// TwinCAT 3 PLC project Untitled1
// ProgramVersion: 3.1.4023.0
// libraries:
//   CmpBitmapPool, * (System)
//   Tc2_MC2, * (Beckhoff Automation GmbH)
//   Tc2_Standard, * (Beckhoff Automation GmbH)
//   Tc2_System, * (Beckhoff Automation GmbH)
//   Tc2_Utilities, * (Beckhoff Automation GmbH)
//   Tc3_Module, * (Beckhoff Automation GmbH)
// project tree:
//   DUTs/ A21ToolStorage.TcDUT (not stored), Bundle.TcDUT (not stored), EOAT.TcDUT (not stored), Interval.TcDUT (not stored), PositionMaterials.TcDUT (not stored)
//   DUTs/Enums/ A21.TcDUT (not stored), Chipboard.TcDUT (not stored), Homing.TcDUT (not stored), SectionEnum.TcDUT (not stored), Surface.TcDUT (not stored), WoodBunk.TcDUT
//   DUTs/Insertion/Drives/ AirPiston.TcPOU, ClearLinkMC.TcPOU (not stored), SimplePiston.TcPOU
//   DUTs/Insertion/ Insertion.TcPOU (not stored), SuctionPad.TcDUT (not stored)
//   DUTs/Insertion/Prototypes/ FBA_Drive.TcPOU (not stored), I_ContinuousDrive.TcIO (not stored), I_Drive.TcIO, I_PositionalDrive.TcIO, I_EncodedDrive.TcIO
//   DUTs/Machines/ Conveyor.TcPOU (not stored), ConveyorMode.TcDUT (not stored), KukaRobot.TcPOU, RobotA21.TcPOU, StrapMachine.TcPOU (not stored)
//   DUTs/Material Holders/ MaterialHolder.TcPOU, SkidMagazine.TcPOU (not stored), StagingTable.TcPOU, MaterialSlot.TcDUT (not stored)
//   GVLs/ StorageArrays.TcGVL, GVL.TcGVL, Hardware.TcGVL (not stored), Misc.TcGVL (not stored)
//   / PlcTask.TcTTO (not stored)
//   POUs/ FB_System.TcPOU (not stored), MAIN.TcPOU (not stored), WoodBunkEx.TcPOU, ChipboardEx.TcPOU (not stored)
//   POUs/Hardware Calls/ InsertionQuality.TcPOU (not stored), CallHardware.TcPOU (not stored), SetSuctions.TcPOU (not stored), SetupHardware.TcPOU
//   POUs/Utility/ AddToStringArray.TcPOU (not stored), BoolVLArrayToInteger.TcPOU (not stored), BoolPtrArrayToInteger.TcPOU (not stored), IntegerBitAccess.TcPOU (not stored), IntegerToBoolArray.TcPOU (not stored), JoinStrings.TcPOU (not stored), WithinTolerance.TcPOU (not stored)
// real-time tasks:
//   TASK PlcTask: cycle T#10ms, priority 20, ADS port 350

// ---- DUTs/Enums/WoodBunk.TcDUT
{attribute 'qualified_only'}
{attribute 'to_string'}
TYPE WoodBunk : //21
(
	NULL, 
	
	WDS08, //side
	WDS10, 
	WDS12, 
	WDS14, 
	
	WDS20, //side - same size as TOP
	WDS22, 
	WDS28, 
	
	WDB20, //bottom
	WDB22, 
	WDB28,

	WDT20, //top
	WDT22, 
	WDT28,
	
	WDW20, //special top (wide) 
	WDW22,
	
	
	size
	(*
	WDS08_WDS08, //side combined - X - 2 wood bunks joined by underscore
	WDS08_WDS10, 
	WDS12_WDS12, 
	WDS12_WDS14, 
	WDS20_WDS10, 
	WDS20_WDS12, 
	
	sizeAll
	*)
);
END_TYPE

// ---- GVLs/StorageArrays.TcGVL
//{attribute 'qualified_only'}
VAR_GLOBAL //data arrays to be passed into material holder FBs - do not access directly
	
	skidSlotsA21Left, skidSlotsA21Right : ARRAY[1..2] OF STRING; //chipboard skid
	skidOccupancyA21Left, skidOccupancyA21Right : ARRAY[1..2] OF BOOL;
	skidHmiA21Left, skidHmiA21Right : ARRAY[1..2] OF MaterialSlot;
	
	magazineSlotsA21Left, magazineSlotsA21Right : ARRAY[1..15] OF STRING; //wood bunk magazine
	magazineOccupancyA21Left, magazineOccupancyA21Right : ARRAY[1..15] OF BOOL;
	magazineHmiA21Left, magazineHmiA21Right : ARRAY[1..15] OF MaterialSlot;
	
	tableSlotsA21Left, tableSlotsA21Right : ARRAY[1..10] OF STRING; //staging table
	tableOccupancyA21Left, tableOccupancyA21Right AT %I* : ARRAY[1..10] OF BOOL;
	tableHmiA21Left, tableHmiA21Right : ARRAY[1..10] OF MaterialSlot;
END_VAR

// ---- GVLs/GVL.TcGVL
{attribute 'qualified_only'}
VAR_GLOBAL CONSTANT
	maxPairs : INT := 16;
	maxQueue : INT := 16;
END_VAR

// ---- DUTs/Insertion/Prototypes/I_Drive.TcIO
INTERFACE I_Drive

{attribute 'monitoring':='call'}
PROPERTY ABSTRACT AtHome : BOOL
GET
END_GET
END_PROPERTY

{attribute 'monitoring':='call'}
PROPERTY ABSTRACT AtInnerLimit : BOOL
GET
END_GET
END_PROPERTY

{attribute 'monitoring':='call'}
PROPERTY ABSTRACT AtOuterLimit : BOOL
GET
END_GET
END_PROPERTY

{attribute 'monitoring':='call'}
PROPERTY ABSTRACT Busy : BOOL
GET
END_GET
END_PROPERTY

{attribute 'monitoring':='call'}
PROPERTY ABSTRACT Contact : BOOL
GET
END_GET
END_PROPERTY

{attribute 'monitoring':='call'}
PROPERTY ABSTRACT Error : BOOL
GET
END_GET
END_PROPERTY

{attribute 'monitoring':='call'}
PROPERTY ABSTRACT HomeSet : BOOL
GET
END_GET
END_PROPERTY

METHOD ABSTRACT homingSequence : BOOL
VAR_INPUT
END_VAR
END_METHOD

METHOD ABSTRACT stop : BOOL
VAR_INPUT
END_VAR
END_METHOD

END_INTERFACE

// ---- DUTs/Insertion/Prototypes/I_PositionalDrive.TcIO
INTERFACE I_PositionalDrive EXTENDS I_Drive

PROPERTY ABSTRACT CurrentPosition : LREAL
GET
END_GET
SET
END_SET
END_PROPERTY

METHOD ABSTRACT moveAbsolute : BOOL
VAR_INPUT
	newTarget : LREAL; 
END_VAR
END_METHOD

METHOD ABSTRACT moveRelative : BOOL
VAR_INPUT
	distance : LREAL;
END_VAR
END_METHOD

PROPERTY ABSTRACT TargetPosition : LREAL
GET
END_GET
SET
END_SET
END_PROPERTY

END_INTERFACE

// ---- DUTs/Insertion/Prototypes/I_EncodedDrive.TcIO
INTERFACE I_EncodedDrive EXTENDS I_PositionalDrive, I_ContinuousDrive
//this drive can perform absolute/relative targeting and continuous motion
//only used if a drive with both encoded and continuous behavior is needed

END_INTERFACE

// ---- DUTs/Insertion/Drives/AirPiston.TcPOU
FUNCTION_BLOCK AirPiston EXTENDS FBA_Drive IMPLEMENTS I_ContinuousDrive
VAR_OUTPUT
	valveExtend AT %Q* : BOOL;
	valveRetract AT %Q* : BOOL;
END_VAR
VAR
	mode : (HOLD, IN, OUT, BRAKE);
	
	useBrake : BOOL; //set to FALSE if retraction brake is not required
	brakePulse : TP; //generates the retraction pulse
END_VAR
VAR_STAT CONSTANT
	brakeTime : TIME := T#650MS;
END_VAR

IF NOT bEnable THEN
	stop();
	RETURN;
END_IF

brakePulse(IN:= , PT:= brakeTime, Q=> , ET=> ); //reversal to act as brake
brakePulse.IN := brakePulse.IN AND brakePulse.Q; //automatically turn off pulse

override(); //alters the mode to prevent exceeding limits

CASE mode OF
	HOLD:
		valveExtend := FALSE;
		valveRetract := FALSE;
		
	IN:
		valveExtend := TRUE;
		valveRetract := FALSE;
		
	OUT:
		valveExtend := FALSE;
		valveRetract := TRUE;
		
	BRAKE: //coasts past inner limit, then slides back
		valveExtend := FALSE;
		valveRetract := TRUE;
		
		IF innerLimit THEN
			mode := HOLD;
		END_IF
		
END_CASE

valveRetract := valveRetract OR brakePulse.Q; //from mode or brake

PROPERTY Busy : BOOL
GET
Busy :=
	mode <> HOLD AND
	valveExtend OR valveRetract;
END_GET
END_PROPERTY

PROPERTY Error : BOOL
GET
END_GET
END_PROPERTY

METHOD extend : BOOL
VAR_INPUT
END_VAR
IF mode <> BRAKE THEN
	mode := IN;
END_IF
END_METHOD

METHOD homingSequence : BOOL
CASE step OF
	Homing.IDLE:
		step := Homing.OUT;
		
	Homing.OUT: //towards home
		mode := OUT;
		
		IF home THEN //if reached home
			step := Homing.DONE;
		END_IF
		
	Homing.DONE:
		mode := HOLD;
		homingComplete := TRUE;
		
		homingSequence := TRUE;		
	
END_CASE
END_METHOD

METHOD moveContinuous : BOOL
VAR_INPUT
	direction : MC_Direction;
END_VAR
IF direction = MC_Positive_Direction THEN
	retract();
ELSIF direction = MC_Negative_Direction THEN
	extend();
END_IF
END_METHOD

METHOD PRIVATE override : BOOL
VAR_INPUT
END_VAR
IF brakePulse.Q THEN
	mode := HOLD;
END_IF

IF home AND_THEN (valveRetract OR mode = OUT) THEN
	mode := HOLD;
	
ELSIF (innerLimit OR contactSensor) AND_THEN (valveExtend OR mode = IN) THEN	
	brakePulse.IN := useBrake;
	mode := HOLD;
END_IF


IF NOT bEnable THEN
	stop();
END_IF
END_METHOD

METHOD retract : BOOL
VAR_INPUT
END_VAR
IF mode <> BRAKE THEN
	mode := OUT;
END_IF
END_METHOD

METHOD stop : BOOL
VAR_INPUT
END_VAR
valveExtend := FALSE;
valveRetract := FALSE;
mode := HOLD;
END_METHOD

END_FUNCTION_BLOCK

// ---- DUTs/Insertion/Drives/SimplePiston.TcPOU
FUNCTION_BLOCK SimplePiston
VAR_INPUT
	bEnable : BOOL;
END_VAR
VAR_OUTPUT
	pistonExtend AT %Q* : BOOL;
	pistonRetract AT %Q* : BOOL;
	
	extended AT %I* : BOOL;
	retracted AT %I* : BOOL;
END_VAR
VAR
	mode : (HOLD, IN, OUT);
END_VAR

IF
	NOT bEnable OR
	(retracted AND_THEN (pistonRetract OR mode = OUT)) OR
	(extended AND_THEN (pistonExtend OR mode = IN))
THEN
	mode := HOLD;
END_IF

CASE mode OF
	HOLD:
		pistonRetract := FALSE;
		pistonExtend := FALSE;
		
	IN:
		pistonRetract := FALSE;
		pistonExtend := TRUE;
	
	OUT:
		pistonRetract := TRUE;
		pistonExtend := FALSE;
	
END_CASE

METHOD extend : BOOL
VAR_INPUT
END_VAR
mode := IN;
END_METHOD

METHOD retract : BOOL
VAR_INPUT
END_VAR
mode := OUT;

retract := retracted;
END_METHOD

METHOD stop : BOOL
VAR_INPUT
END_VAR
pistonExtend := FALSE;
pistonRetract := FALSE;
mode := HOLD;
END_METHOD

END_FUNCTION_BLOCK

// ---- DUTs/Machines/KukaRobot.TcPOU
FUNCTION_BLOCK KukaRobot
VAR_OUTPUT
	forceStop AT %Q* : BOOL;
	resetSignal AT %Q* : BOOL;
	
	offline AT %I* : BOOL;
	operational : BOOL;
	reservation : INT := SectionEnum.NULL_SECTION;
	
	error : BOOL;
	errId : DINT;
	
	outputs AT %Q* : ARRAY[1..50] OF WORD;
	inputs AT %I* : ARRAY[1..20] OF WORD;
END_VAR
VAR
	hmiReservation : STRING;
END_VAR
(*
generic KUKA robot with 50 WORD outputs and 20 WORD inputs
includes minimal diagnostics to detect if robot is offline
robots should always be reserved before sending a task
*)

operational := NOT offline;

error := offline; //add any addition conditions with OR

//{attribute 'monitoring' := 'variable'}
{attribute 'monitoring' := 'call'}
PROPERTY Busy : BOOL
GET
END_GET
END_PROPERTY

METHOD clearCommand : BOOL
VAR_INPUT
END_VAR
MEMSET(ADR(outputs), 0, SIZEOF(outputs));
END_METHOD

//{attribute 'monitoring' := 'variable'}
{attribute 'monitoring' := 'call'}
PROPERTY Done : BOOL
GET
END_GET
END_PROPERTY

METHOD eStop : BOOL
VAR_INPUT
END_VAR
forceStop := TRUE;
eStop := TRUE;
END_METHOD

METHOD fullCommand : BOOL
VAR_INPUT
	newOutputs : REFERENCE TO ARRAY[1..50] OF WORD;
END_VAR
//IF NOT Busy THEN
	//RETURN;
//END_IF

outputs := newOutputs;
fullCommand := Done;

(*
CASE step OF
	SEND_COMMAND: //wait 1 cycle
		outputs := newOutputs;
		step := WAIT;
		
	WAIT:
		IF done THEN
			(*	
			IF NOT reset() THEN
				RETURN;
			END_IF
			
			step := 0;
			*)
			setCommandAndWait := TRUE;
		END_IF
		
END_CASE
*)
END_METHOD

{attribute 'monitoring' := 'call'}
PROPERTY Ready : BOOL
GET
END_GET
END_PROPERTY

METHOD release : BOOL
VAR_INPUT
	reservee : INT;
END_VAR
IF reservation = reservee THEN
	reservation := SectionEnum.NULL_SECTION;
	release := TRUE;
END_IF
END_METHOD

METHOD reserve : BOOL
VAR_INPUT
	reservee : INT;
END_VAR
(*
this method exists because chipboard and wood bunk operations use the same robot
both sections need to check if the robot is open to commands before use
*)
IF Reserved AND reservation = reservee THEN
	reserve := TRUE;

ELSIF NOT Reserved THEN
	reservation := reservee;
	reserve := TRUE;

END_IF
END_METHOD

{attribute 'monitoring' := 'call'}
PROPERTY Reserved : BOOL
GET
Reserved := reservation <> SectionEnum.NULL_SECTION;
END_GET
END_PROPERTY

METHOD reset : BOOL
//resetSignal := TRUE;
//done := FALSE;

MEMSET(ADR(outputs), 0, SIZEOF(outputs));
(*
IF ready AND completedTask = 0 THEN
	resetSignal := FALSE;
	reset := TRUE;
END_IF
*)
END_METHOD

METHOD resume : BOOL
VAR_INPUT
END_VAR
forceStop := FALSE;

resume := NOT error AND errId = 0;
END_METHOD

METHOD setGroup : BOOL
VAR_INPUT
	group : INT;
	value : INT;
END_VAR
{warning disable C0195}
outputs[group] := value;
END_METHOD

END_FUNCTION_BLOCK

// ---- DUTs/Machines/RobotA21.TcPOU
FUNCTION_BLOCK RobotA21 EXTENDS KukaRobot
VAR_OUTPUT //from outputs array
	{warning disable C0195}
	taskID : A21;
	param1 : INT;
	param2 : INT;
	Xmm : INT;
	Ymm : INT;
	Zmm : INT;
	angle : INT;
	stagingOccupancy : INT;
	insertionSuctionStatus : INT;
	magazineStatus : INT; //unused
	inspectionValue : INT;
	
	strapSafetyOut : BOOL;
END_VAR
VAR_OUTPUT //from inputs array
	tool : SectionEnum := SectionEnum.WOOD_BUNK;
	suspendedMaterial : STRING;
	//gripper : EOAT := (id := SectionEnum.WOOD_BUNK, material := '');
	
	completedTask : A21;
	eoatDistance : INT;
	woodBunkAvailability : INT;
	chipboardAvailability : INT;
	materialAtHoldingPosition : INT;
	
	strapSafetyIn : BOOL;
END_VAR
VAR
	reservationEnum : SectionEnum;
	hmiTask : STRING;
	hmiTool : STRING;
END_VAR
(*
extends KukaRobot
assigns descriptive labels to each IO group from the array
additional section-specific methods to get/set IO groups
*)

(*
parameters - aliases to IO elements
command - full IO array
*)
{warning disable C0195}
SUPER^();

strapSafetyOut := NOT strapperA21.enable AND NOT strapperA21.execute;
outputs[8].15 := strapSafetyOut;

outputs[1] := taskID;
outputs[2] := param1;
outputs[3] := param2;
outputs[4] := Xmm;
outputs[5] := Ymm;
outputs[6] := Zmm;
outputs[7] := angle;
outputs[8] := stagingOccupancy;
outputs[9] := insertionSuctionStatus;
outputs[10] := magazineStatus;
outputs[11] := inspectionValue;

outputs[8].15 := strapSafetyOut;

refreshParameters();

reservationEnum := reservation;
IF reservationEnum = SectionEnum.NULL_SECTION THEN
	hmiReservation := 'N/A';
ELSE
	hmiReservation := TO_STRING(reservationEnum);
END_IF

hmiTask := TO_STRING(taskID);
hmiTool := TO_STRING(tool);

{attribute 'monitoring' := 'call'}
PROPERTY Busy : BOOL
GET
VAR
	//emptyOutput : ARRAY[1..50] OF INT;
END_VAR
//Busy stays TRUE until outputs are cleared AND completed task has elapsed
//Ready is always inverse of Busy
refreshParameters();

Busy := taskID <> 0 OR completedTask <> 0;
END_GET
END_PROPERTY

METHOD changeEOAT : BOOL
VAR_INPUT
	targetTool : SectionEnum;
END_VAR
setGroup(group := 1, value := A21.TOOL_CHANGE_CHIPBOARD);
setGroup(group := 1, value := A21.TOOL_CHANGE_BUNK);

changeEOAT := tool = targetTool;
END_METHOD

METHOD clearCommand : BOOL
VAR_INPUT
END_VAR
SUPER^.clearCommand();

refreshParameters();
END_METHOD

{attribute 'monitoring' := 'call'}
PROPERTY Done : BOOL
GET
refreshParameters();

Done :=
	completedTask = taskID AND
	taskID <> 0 AND
	completedTask <> 0;
END_GET
END_PROPERTY

{attribute 'monitoring' := 'call'}
PROPERTY HoldMaterial : STRING
GET
HoldMaterial := suspendedMaterial;
END_GET
SET
suspendedMaterial := HoldMaterial;
END_SET
END_PROPERTY

{attribute 'monitoring' := 'call'}
PROPERTY Ready : BOOL
GET
refreshParameters();

Ready := taskID = 0 AND completedTask = 0;
END_GET
END_PROPERTY

METHOD PRIVATE refreshParameters : BOOL
VAR_INPUT
END_VAR
{warning disable C0196}
taskID := outputs[1];
param1 := outputs[2];
param2 := outputs[3];
Xmm := outputs[4];
Ymm := outputs[5];
Zmm := outputs[6];
angle := outputs[7];
stagingOccupancy := outputs[8];
insertionSuctionStatus := outputs[9];
magazineStatus := outputs[10]; //unused
inspectionValue := outputs[11];

completedTask := inputs[1];
eoatDistance := inputs[2];
woodBunkAvailability := inputs[3];
chipboardAvailability := inputs[4];
materialAtHoldingPosition := inputs[5];
//robotEOAT := inputs[6];

strapSafetyIn := inputs[4].15;
END_METHOD

METHOD setGroup : BOOL
VAR_INPUT
	group : INT;
	value : INT;
END_VAR
SUPER^.setGroup(group := group, value := value);

refreshParameters();
END_METHOD

METHOD setParameters : BOOL
VAR_INPUT
	newTaskID : INT;
	newParam1 : INT;
	newParam2 : INT;
	newXmm : INT;
	newYmm : INT;
	newZmm : INT;
	newAngle : INT;
	newStagingOccupancy : INT;
	newInsertionSuctionStatus : INT;
	newMagazineStatus : INT; //unused
	newInspectionValue : INT;
END_VAR
setGroup(group := 1, value := newTaskID);
setGroup(group := 2, value := newParam1);
setGroup(group := 3, value := newParam2);
setGroup(group := 4, value := newXmm);
setGroup(group := 5, value := newYmm);
setGroup(group := 6, value := newZmm);
setGroup(group := 7, value := newAngle);

newStagingOccupancy.15 := NOT strapperA21.enable AND NOT strapperA21.execute;
setGroup(group := 8, value := newStagingOccupancy);

setGroup(group := 9, value := newInsertionSuctionStatus);
setGroup(group := 10, value := newMagazineStatus);
setGroup(group := 11, value := newInspectionValue);

refreshParameters();
END_METHOD

END_FUNCTION_BLOCK

// ---- DUTs/Material Holders/MaterialHolder.TcPOU
FUNCTION_BLOCK MaterialHolder
VAR_IN_OUT
	slots : ARRAY[*] OF STRING;
	occupied : ARRAY[*] OF BOOL;
	
	hmiTable : ARRAY[*] OF MaterialSlot;
END_VAR
VAR
	numSlots : INT;
END_VAR

(*
by default:
	hmiTable contains the true data, including IO mapped to hardware
	slots and occupied cyclically copy data from hmiTable

if hmiTable is NULL (not passed in), then slots and occupied will store the true data
	
the program will access data using slots/occupied via methods
when the data is changed, data is copied from slots/occupied to hmiTable

this ensures that the methods update the HMI, and the HMI updates the data
*)


IF hmiTable <> 0 AND_THEN (slots <> 0  AND occupied <> 0) THEN
	writeArrays();
END_IF

numSlots := TO_INT(UPPER_BOUND(slots, 1) - LOWER_BOUND(slots, 1) + 1);

METHOD clear : BOOL
VAR_INPUT
END_VAR
MEMSET(ADR(slots), 0, SIZEOF(slots));
END_METHOD

METHOD findSlot : BOOL
VAR_INPUT
	materialID : STRING;
END_VAR
VAR_OUTPUT
	atPosition : INT := -1;
END_VAR
VAR
	i : INT;
END_VAR
(*
IF materialID = '' THEN
	RETURN;
END_IF
*)
FOR i:=1 TO GVL.maxQueue BY 1 DO
	IF slots[i] = materialID THEN
		atPosition := i;
		findSlot := TRUE;
		RETURN;
	END_IF
END_FOR
END_METHOD

METHOD getSlot : STRING
VAR_INPUT
	i : DINT;
END_VAR
VAR_OUTPUT
	errorBounds : BOOL;
END_VAR
errorBounds := i < LOWER_BOUND(slots, 1) OR i > UPPER_BOUND(slots, 1);

IF errorBounds THEN
	RETURN;
END_IF

getSlot := slots[i];
END_METHOD

METHOD getSlotsAsArray : POINTER TO STRING
getSlotsAsArray := ADR(slots);
END_METHOD

METHOD isOccupied : BOOL
VAR_INPUT
	i : DINT;
END_VAR
VAR_OUTPUT
	errorBounds : BOOL;
END_VAR
errorBounds := i < LOWER_BOUND(slots, 1) OR i > UPPER_BOUND(slots, 1);

IF errorBounds THEN
	RETURN;
END_IF

isOccupied := occupied[i];
END_METHOD

METHOD setSlots : BOOL
VAR_IN_OUT
	newSlots : ARRAY[*] OF STRING;
END_VAR
VAR
	i : DINT;
	j : DINT;
END_VAR
{warning disable C0195}
setSlots := MEMCPY(
	slots, 
	newSlots, 
	SIZEOF(STRING) * MIN(
		(1 + UPPER_BOUND(newSlots, 1) - LOWER_BOUND(newSlots, 1)),
		(1 + UPPER_BOUND(slots, 1) - LOWER_BOUND(slots, 1))
	)) > 0;
	
IF hmiTable <> 0 THEN
	writeHmiTable();
END_IF
END_METHOD

METHOD PROTECTED writeArrays : BOOL
VAR
	i : DINT;
END_VAR
FOR i:=LOWER_BOUND(hmiTable, 1) TO UPPER_BOUND(hmiTable, 1) BY 1 DO
	slots[i] := hmiTable[i].material;
	occupied[i] := hmiTable[i].occupied;
END_FOR
END_METHOD

METHOD PROTECTED writeHmiTable : BOOL
VAR
	i : DINT;
END_VAR
FOR i:=LOWER_BOUND(hmiTable, 1) TO UPPER_BOUND(hmiTable, 1) BY 1 DO
	hmiTable[i].material := slots[i];
	hmiTable[i].occupied := occupied[i];
END_FOR
END_METHOD

END_FUNCTION_BLOCK

// ---- DUTs/Material Holders/StagingTable.TcPOU
FUNCTION_BLOCK StagingTable EXTENDS MaterialHolder

SUPER^();

METHOD autofill : BOOL
VAR_INPUT
	materialID : STRING;
END_VAR
VAR_OUTPUT
	slot : INT;
END_VAR
VAR
	i : INT;
END_VAR
(*
this method will automatically find an open slot
*)
IF isFull() OR materialID = '' THEN
	RETURN;
END_IF

IF findOpenSlot(materialID, openSlot=> slot) THEN
	place(slot, materialID);
	autofill := TRUE;
END_IF

IF hmiTable <> 0 THEN
	writeHmiTable();
END_IF
END_METHOD

METHOD findOpenSlot : BOOL
VAR_INPUT
	materialID : STRING;
END_VAR
VAR_OUTPUT
	openSlot : INT := 0;
END_VAR
VAR
	i : INT;
END_VAR
IF FIND(materialID, 'WDW') > 0 THEN //top wide, load in slot 9-10
	FOR i:=9 TO 10 BY 1 DO
		IF slots[i] = '' THEN
			findOpenSlot := TRUE;
			openSlot := i;
			RETURN;
		END_IF
	END_FOR
	
//ELSIF FIND(materialID, 'WDT') > 0 OR FIND(materialID, 'WDS') > 0 THEN //standard width, load in slot 3-10
ELSIF FIND(materialID, 'WD') > 0 THEN //standard width, load in slot 1-8
	FOR i:=1 TO 8 BY 1 DO
		IF slots[i] = '' THEN
			findOpenSlot := TRUE;
			openSlot := i;
			RETURN;
		END_IF
	END_FOR
	
END_IF
END_METHOD

METHOD isEmpty : BOOL
VAR
	i : INT;
	temp : BOOL;
END_VAR
FOR i:=1 TO numSlots BY 1 DO
	temp := temp OR occupied[i]; //TRUE if any slots are occupied
END_FOR

isEmpty := NOT temp; //invert result - FALSE if any slots are occupied
END_METHOD

METHOD isFull : BOOL
VAR
	i : INT;
	temp : BOOL := TRUE;
END_VAR
FOR i:=1 TO numSlots BY 1 DO
	temp := temp AND occupied[i];
END_FOR

isFull := temp;
END_METHOD

METHOD place : BOOL
VAR_INPUT
	i : INT;
	materialID : STRING;
END_VAR
IF slots[i] = '' THEN
	slots[i] := materialID;
	place := TRUE;
END_IF

IF hmiTable <> 0 THEN
	writeHmiTable();
END_IF
END_METHOD

METHOD remove : BOOL
VAR_INPUT
	i : INT;
END_VAR
VAR_OUTPUT
	materialID : STRING;
END_VAR
remove := slots[i] <> '';

materialID := slots[i];
slots[i] := '';

IF hmiTable <> 0 THEN
	writeHmiTable();
END_IF
END_METHOD

END_FUNCTION_BLOCK

// ---- POUs/Hardware Calls/SetupHardware.TcPOU
FUNCTION SetupHardware : BOOL
VAR
	iWoodBunkSlot : WoodBunk;
	iChipboardSlot : Chipboard;
	
	slotsArr : ARRAY[1..GVL.maxQueue] OF STRING;
	
	i : INT;
END_VAR

FOR iWoodBunkSlot:=1 TO WoodBunk.size-1 BY 1 DO //init wood bunk magazine slots
	magazineA21Left.setSlot(i := iWoodBunkSlot, material := TO_STRING(iWoodBunkSlot), error => );
	magazineA21Right.setSlot(i := iWoodBunkSlot, material := TO_STRING(iWoodBunkSlot), error => );
END_FOR

//--------------------------------------------------

FOR iChipboardSlot:=1 TO Chipboard.size-1 BY 1 DO //init chipboard skid slots
	skidA21Left.setSlot(i := iChipboardSlot, material := TO_STRING(iChipboardSlot), error => );
	skidA21Right.setSlot(i := iChipboardSlot, material := TO_STRING(iChipboardSlot), error => );
END_FOR

//--------------------------------------------------

FOR i:=1 TO GVL.maxQueue BY 1 DO //get wood bunk magazine + chipboard skid availability from robot1 and robot2
	{warning disable C0195}
	skidA21Left.setOccupancy( i := i, occupancy := IntegerBitAccess(robot1.inputs[4], i-1) );
	skidA21Right.setOccupancy( i := i, occupancy := IntegerBitAccess(robot2.inputs[4], i-1) );

	magazineA21Left.setOccupancy( i := i, occupancy := IntegerBitAccess(robot1.inputs[3], i-1) );
	magazineA21Right.setOccupancy( i := i, occupancy := IntegerBitAccess(robot2.inputs[3], i-1) );
END_FOR

//--------------------------------------------------

//enable all drives
verticalDriveA21Left.bEnable := 
verticalDriveA21Right.bEnable := 
horizontalDriveA21Left.bEnable := 
horizontalDriveA21Right.bEnable := 
pistonA21Bottom.bEnable := 
TRUE;

END_FUNCTION

// ---- POUs/WoodBunkEx.TcPOU
FUNCTION_BLOCK WoodBunkEx
VAR_IN_OUT //controls
	execute : BOOL;
	stop : BOOL;
	
	manualStep : BOOL;
	manualSuction : BOOL;
END_VAR
VAR_IN_OUT //references to required hardware
	robotLeft, robotRight : RobotA21;
	toolStorageLeft, toolStorageRight : A21ToolStorage;
	
	stagingTableLeft, stagingTableRight : StagingTable;
	magazineLeft, magazineRight : SkidMagazine;
	
	strapper : StrapMachine;
	
	horizontalDriveLeft, horizontalDriveRight : AirPiston;
	verticalDriveLeft, verticalDriveRight : ClearLinkMC;
	pistonBottom : SimplePiston;
	
	suctionTop : ARRAY[*] OF SuctionPad; (*1..3*)
	suctionLeft : ARRAY[*] OF SuctionPad; (*1..4*)
	suctionRight : ARRAY[*] OF SuctionPad; (*1..4*)
	suctionBottom : ARRAY[*] OF SuctionPad; (*1..2*)
END_VAR
VAR_OUTPUT
	//ready : BOOL;
	done : BOOL;
	
	generalError : BOOL;
	errorLeft, errorRight : BOOL;
END_VAR
VAR //for testing, to be removed when deployoed
	latchLeft, latchRight : BOOL; //prevents SMC sliders from overshooting the inner limit sensor
	
	suctionEnableTop : BOOL;
	suctionEnableLeft : BOOL;
	suctionEnableRight : BOOL;
	suctionEnableBottom : BOOL;
END_VAR
VAR	
	topSuctionDelay : TON;
	
	step : (IDLE, STAGING, LOAD_WB, PUSH, STRAP, RELEASE, COMPLETE := 1050);
	iPair : INT;
	//these 2 ints should replace the 4 ints after
	masterStep : INT;
	subStepLeft, subStepRight : INT;
	
	loadSet : INT;
	loadStepLeft, loadStepRight : INT;
	
	stageSet : INT;	
	stageStepLeft, stageStepRight : INT;
	iSlotLeft, iSlotRight : INT;
END_VAR
VAR //local types
	demoHeight : REAL := 600; //mm
	materialsArr : ARRAY[0..GVL.maxPairs] OF PositionMaterials := [
		(
			position := 0,
			top := 'WDS20', left := 'WDS20', right := 'WDS20', bottom := 'WDB20'
		),
		(
			position := 69,
			top := 'WDS20', left := 'WDS20', right := 'WDS20', bottom := 'WDB20'
		)];
	
	templateSlotsLeft, templateSlotsRight : ARRAY[1..10] OF STRING;
	templateOccupancyLeft, templateOccupancyRight : ARRAY[1..10] OF BOOL;
	stagingTemplateLeft, stagingTemplateRight AT %M* : StagingTable;	
	stagingArrayLeft, stagingArrayRight : ARRAY[0..(GVL.maxPairs+1)*2] OF STRING;
	
	insertionLeft, insertionRight : Insertion;
	loadedMaterials : ARRAY[Surface.TOP..Surface.BOTTOM] OF STRING;
END_VAR
VAR CONSTANT
	sectionID : SectionEnum := SectionEnum.WOOD_BUNK;
END_VAR
VAR
	a,b,c,d : BOOL;
	suctionTimerLeft, suctionTimerRight : TON;
END_VAR

callLocalModules(); //initialize local modules

IF stop THEN
	stopSequence(); //stop everything
	RETURN;
END_IF

IF NOT insertionLeft.screw.HomeSet AND insertionRight.screw.HomeSet THEN
	homingSequence(); //homing all motion devices and robots
	RETURN;
END_IF

a S= suctionTop[1].occupied AND suctionTop[2].occupied AND suctionTop[3].occupied;
b S= suctionLeft[1].occupied AND suctionLeft[2].occupied AND suctionLeft[3].occupied AND suctionLeft[4].occupied;
c S= suctionRight[1].occupied AND suctionRight[2].occupied AND suctionRight[3].occupied AND suctionRight[4].occupied;
d S= suctionBottom[1].occupied AND suctionBottom[2].occupied;

CASE step OF
	IDLE:
		IF execute THEN
			execute := FALSE;
			suctionEnableTop := suctionEnableLeft := suctionEnableRight := suctionEnableBottom := FALSE;
			step := STAGING;
		END_IF
		
		SetSuctions(suctionTop, suctionEnableTop);
		SetSuctions(suctionLeft, suctionEnableLeft);
		SetSuctions(suctionRight, suctionEnableRight);
		SetSuctions(suctionBottom, suctionEnableBottom);
		
	STAGING:
		IF NOT done THEN
			done := stage(error => generalError);
		END_IF
		
		IF
			(manualStep AND_THEN execute) OR
			(NOT manualStep AND_THEN done)
		THEN
			execute := FALSE;
			done := FALSE;
			step := LOAD_WB;
		END_IF
	
	LOAD_WB:
		IF NOT done THEN
			done := load(pairIndex := iPair, error => generalError);
		END_IF
		
		IF manualSuction THEN
			SetSuctions(suctionTop, suctionEnableTop);
			SetSuctions(suctionLeft, suctionEnableLeft);
			SetSuctions(suctionRight, suctionEnableRight);
			SetSuctions(suctionBottom, suctionEnableBottom);
		END_IF
		
		IF
			(manualStep AND_THEN execute) OR
			(NOT manualStep AND_THEN done)
		THEN
			done := FALSE;
			suctionEnableTop := suctionEnableLeft := suctionEnableRight := suctionEnableBottom := FALSE;
			execute := FALSE;
			
			step := PUSH;
		END_IF
		
	PUSH:
		IF
			(manualStep AND_THEN execute) OR
			(latchLeft AND latchRight AND pistonBottom.extended)
		THEN
			latchLeft := latchRight := FALSE;
			execute := FALSE;
			step := STRAP;
		END_IF
		
		IF NOT validateSuctionQuality(checkTop:= TRUE, checkLeft:= TRUE, checkRight:= FALSE, checkBottom:= FALSE) THEN
			generalError := TRUE;
			RETURN;
		END_IF
		(*
		IF 
			insertionLeft.sliderPos <> demoHeight/2 //OR 
			//insertionRight.sliderPos <> demoHeight/2 //OR 
			//NOT insertionBottom.contact
		THEN
			insertionLeft.slideAbsolute(demoHeight/2);
			//insertionRight.slideAbsolute(demoHeight/2);
			RETURN;
		END_IF
		*)
		
		IF insertionLeft.screw.AtInnerLimit THEN
			latchLeft := TRUE;
		ELSIF NOT latchLeft THEN
			insertionLeft.press();
		END_IF
		
		IF insertionRight.screw.AtInnerLimit THEN
			latchRight := TRUE;
		ELSIF NOT latchRight THEN
			insertionRight.press();
		END_IF
		pistonBottom.extend();
		
	STRAP:
		topSuctionDelay(IN:= , PT:= T#1S, Q=> , ET=> );
		
		strapper.bEnable := TRUE;
		IF strapper.done THEN
			topSuctionDelay.IN := FALSE;
			step := RELEASE;
			RETURN;
		END_IF
		
		IF topSuctionDelay.Q THEN
			SetSuctions(suctionTop, FALSE);
			SetSuctions(suctionLeft, FALSE);
			SetSuctions(suctionRight, FALSE);
			SetSuctions(suctionBottom, FALSE);
		ELSIF strapper.atBundleLevel THEN
			topSuctionDelay.IN := TRUE;
		END_IF
		
		IF strapper.ready THEN
			strapper.strap();
		END_IF
		
		IF execute THEN
			topSuctionDelay.IN := FALSE;
			execute := FALSE;
			step := RELEASE;
		END_IF
		
	RELEASE: //release command		
		//insertionLeft.slideAbsolute(0);
		//insertionRight.slideAbsolute(0);
		
		insertionLeft.release();
		insertionRight.release();
		pistonBottom.retract();
		
		IF 
			(insertionLeft.screw.AtHome AND insertionRight.screw.AtHome AND pistonBottom.retracted) OR
			execute
		THEN
			execute := FALSE;
			step := COMPLETE;
		END_IF
	
	COMPLETE:
		//reset everything
		iPair := (iPair + 1) MOD GVL.maxPairs;
		step := IDLE;
		a := b := c := d := FALSE;
END_CASE

ACTION callLocalModules:
{warning disable C0371}
stagingTemplateLeft(slots := templateSlotsLeft, occupied := templateOccupancyLeft);
stagingTemplateRight(slots := templateSlotsRight, occupied := templateOccupancyRight);

insertionLeft(
	enable:= TRUE, 
	slider:= verticalDriveLeft, 
	screw:= horizontalDriveLeft, 
	contact=> , 
	softContact=> , 
	busy=> , 
	error=> , 
	home=> , 
	homingComplete=> , 
	sliderPos=> );
	
insertionRight(
	enable:= TRUE, 
	slider:= verticalDriveRight, 
	screw:= horizontalDriveRight,  
	contact=> , 
	softContact=> , 
	busy=> , 
	error=> , 
	home=> , 
	homingComplete=> , 
	sliderPos=> );
END_ACTION

METHOD createStagingArrayLeft : BOOL
VAR
	remainingMaterial : STRING;
	splitMaterial : STRING;
	
	i : INT;
END_VAR
FOR i:=0 TO GVL.maxPairs BY 1 DO
	remainingMaterial := materialsArr[i].top;
	WHILE FIND(remainingMaterial, '_') > 0 DO
		splitCombinedMaterials(remainingMaterial, splitMaterial);
		IF splitMaterial <> '' THEN
			AddToStringArray(arr := stagingArrayLeft, newString := splitMaterial, numElements => , nextIndex => );
		END_IF
	END_WHILE
	
	IF remainingMaterial <> '' THEN
		AddToStringArray(arr := stagingArrayLeft, newString := remainingMaterial, numElements => , nextIndex => );
	END_IF
	
	
	remainingMaterial := materialsArr[i].left;
	WHILE FIND(remainingMaterial, '_') > 0 DO
		splitCombinedMaterials(remainingMaterial, splitMaterial);
		IF splitMaterial <> '' THEN
			AddToStringArray(arr := stagingArrayLeft, newString := splitMaterial, numElements => , nextIndex => );
		END_IF
	END_WHILE
	
	IF remainingMaterial <> '' THEN
		AddToStringArray(arr := stagingArrayLeft, newString := remainingMaterial, numElements => , nextIndex => );
	END_IF
END_FOR
END_METHOD

METHOD createStagingArrayRight : BOOL
VAR
	remainingMaterial : STRING;
	splitMaterial : STRING;
	
	i : INT;
END_VAR
FOR i:=0 TO GVL.maxPairs*2 BY 1 DO
	remainingMaterial := materialsArr[i].bottom;
	WHILE FIND(remainingMaterial, '_') > 0 DO
		splitCombinedMaterials(remainingMaterial, splitMaterial);
		IF splitMaterial <> '' THEN
			AddToStringArray(arr := stagingArrayRight, newString := splitMaterial, numElements => , nextIndex => );
		END_IF
	END_WHILE
	
	IF remainingMaterial <> '' THEN
		AddToStringArray(arr := stagingArrayRight, newString := remainingMaterial, numElements => , nextIndex => );
	END_IF
	
	
	
	remainingMaterial := materialsArr[i].right;
	WHILE FIND(remainingMaterial, '_') > 0 DO
		splitCombinedMaterials(remainingMaterial, splitMaterial);
		IF splitMaterial <> '' THEN
			AddToStringArray(arr := stagingArrayRight, newString := splitMaterial, numElements => , nextIndex => );
		END_IF
	END_WHILE
	
	IF remainingMaterial <> '' THEN
		AddToStringArray(arr := stagingArrayRight, newString := remainingMaterial, numElements => , nextIndex => );
	END_IF
END_FOR
END_METHOD

METHOD PROTECTED generateStagingTemplate : BOOL
VAR
	remainingMaterial : STRING;
	splitMaterial : STRING;
	
	i : INT;
END_VAR
VAR_STAT
	temp : INT;
END_VAR
createStagingArrayLeft();
createStagingArrayRight();

//AddToStringArray(arr := stagingArrayLeft, newString := 'WDB20', numElements =>, nextIndex => );

(*
iterate through all pairs and autofill the template
replace succesfully autofilled materials with empty string

when staging needs to be performed a 2nd time, autofilling empty strings is always unsuccessful
*)
FOR i:=0 TO GVL.maxPairs*2 BY 1 DO
	IF stagingTemplateLeft.autofill(materialID := stagingArrayLeft[i]) THEN
		stagingArrayLeft[i] := '';
	END_IF
	
	IF stagingTemplateRight.autofill(materialID := stagingArrayRight[i]) THEN
		stagingArrayRight[i] := '';
	END_IF
END_FOR

(*
stagingTemplateLeft.autofill(demoPairWB.top);
stagingTemplateLeft.autofill(demoPairWB.left);

stagingTemplateRight.autofill(demoPairWB.right);
stagingTemplateRight.autofill(demoPairWB.bottom);
*)

generateStagingTemplate := TRUE;
END_METHOD

ACTION homingSequence:
insertionLeft.homingSequence();
insertionRight.homingSequence();
pistonBottom.retract();
END_ACTION

METHOD PROTECTED load : BOOL
VAR_INPUT
	pairIndex : INT;
END_VAR
VAR_OUTPUT
	error : BOOL;
END_VAR
VAR
	pair : REFERENCE TO PositionMaterials REF= materialsArr[pairIndex];
END_VAR
{warning disable C0371}

IF robotLeft.error OR robotRight.error THEN
	error := TRUE;
	RETURN;
	
ELSIF NOT robotLeft.reserve(sectionID) OR NOT robotRight.reserve(sectionID) THEN //loading requires both robots be reserved together
	RETURN;
	
ELSIF //robots have wrong tool
	(robotLeft.tool <> sectionID AND_THEN NOT robotLeft.changeEOAT(targetTool := sectionID)) OR
	(robotRight.tool <> sectionID AND_THEN NOT robotRight.changeEOAT(targetTool := sectionID))
THEN
	RETURN;
END_IF

CASE loadSet OF
	0: //top and bottom
		IF 
			loadingSequence(
				robot:= robotLeft, 
				table:= stagingTableLeft, 
				loadStep:= loadStepLeft, 
				slot:= iSlotLeft,
				suctions:= suctionTop,
				suctionTimer:= suctionTimerLeft,
				surfaceID:= Surface.TOP, 
				material:= pair.top, 
				fail=> errorLeft)
			
			AND
			loadingSequence(
				robot:= robotRight,
				table:= stagingTableRight, 
				loadStep:= loadStepRight, 
				slot:= iSlotRight,
				suctions:= suctionBottom,
				suctionTimer:= suctionTimerRight,
				surfaceID:= Surface.BOTTOM, 
				material:= pair.bottom, 
				fail=> errorRight)
			
		THEN
			suctionTimerLeft.IN := suctionTimerRight.IN := FALSE;
			loadStepLeft := loadStepRight := 0;
			loadSet := 10;
		END_IF
		
	10: //sides
		IF
			loadingSequence(
				robot:= robotLeft, 
				table:= stagingTableLeft, 
				loadStep:= loadStepLeft, 
				slot:= iSlotLeft,
				suctions:= suctionLeft,
				suctionTimer:= suctionTimerLeft,
				surfaceID:= Surface.LEFT, 
				material:= pair.left, 
				fail=> errorLeft)
			
			AND
			loadingSequence(
				robot:= robotRight, 
				table:= stagingTableRight, 
				loadStep:= loadStepRight, 
				slot:= iSlotRight,
				suctions:= suctionRight,
				suctionTimer:= suctionTimerRight,
				surfaceID:= Surface.RIGHT, 
				material:= pair.right, 
				fail=> errorRight)
		THEN
			suctionTimerLeft.IN := suctionTimerRight.IN := FALSE;
			loadStepLeft := loadStepRight := 0;
			loadSet := COMPLETE;
		END_IF
		
	COMPLETE:
		suctionTimerLeft.IN := suctionTimerRight.IN := FALSE;
		
		loadSet := 0;
		loadStepLeft := loadStepRight := 0;
		
		robotLeft.release(sectionID);
		robotRight.release(sectionID);
		
		load := TRUE;
END_CASE
END_METHOD

METHOD loadingSequence : BOOL
VAR_IN_OUT
	robot : RobotA21;
	table : StagingTable;
	suctions : ARRAY[*] OF SuctionPad;
	loadStep : INT;
	slot : INT;
	
	suctionTimer : TON;
END_VAR
VAR_INPUT
	surfaceID : Surface;
	material : STRING;
END_VAR
VAR_OUTPUT
	fail : BOOL;
END_VAR
VAR
	recoveryMagazine : REFERENCE TO SkidMagazine;
	recoveryStageStep : REFERENCE TO INT;
	suctionDelay : TIME := T#2S;
END_VAR
{warning disable C0371}
IF material = '' THEN
	robot.clearCommand();
	loadingSequence := TRUE;
	RETURN;
END_IF

CASE loadStep OF
	0: //wait for robot
		robot.clearCommand();
		IF robot.Ready THEN
			loadStep := 10;
			slot := 0;
		END_IF
		
	10: //grab from table
		IF slot < 1 AND_THEN NOT table.findSlot(materialID := material, atPosition => slot) THEN 
			fail := TRUE;
			RETURN;
		END_IF
		
		IF NOT table.isOccupied(i := slot) AND table.getSlot(i := slot) <> '' THEN //move from table to robot gripper
			robot.HoldMaterial := table.getSlot(i := slot);
			table.remove(i := slot, materialID => );
		END_IF
		
		IF robot.Done THEN
			loadStep := COMPLETE;
			RETURN;
		ELSIF robot.materialAtHoldingPosition >= 1 AND robot.materialAtHoldingPosition <= 8 THEN
			loadStep := 20;
			RETURN;
		END_IF
		
		CASE surfaceID OF
			Surface.TOP: 					robot.setGroup(group := 1, value := A21.LOAD_BUNK_TOP); 
			Surface.LEFT, Surface.RIGHT: 	robot.setGroup(group := 1, value := A21.LOAD_BUNK_SIDE);
			Surface.BOTTOM: 				robot.setGroup(group := 1, value := A21.LOAD_BUNK_BOTTOM);
		END_CASE
		robot.setGroup(group := 2, value := slot); 
			
	20: //place to insertion
		IF robot.materialAtHoldingPosition > 0 AND robot.HoldMaterial <> '' THEN //move from gripper to insertion
			IF loadedMaterials[surfaceID] = '' THEN //transfer to insertion as is
				loadedMaterials[surfaceID] := robot.HoldMaterial;
			ELSE //join with existing material using underscore _
				loadedMaterials[surfaceID] := JoinStrings(loadedMaterials[surfaceID], robot.HoldMaterial, '_');
			END_IF
			robot.HoldMaterial := '';
		END_IF
		
		CASE surfaceID OF
			Surface.TOP, Surface.BOTTOM:
				SetSuctions(suctions, TRUE (*robot.materialAtHoldingPosition = 1 OR robot.materialAtHoldingPosition = 4*));
				
			Surface.LEFT, Surface.RIGHT:
				SetSuctions(suctions, TRUE (*robot.materialAtHoldingPosition = 2 OR robot.materialAtHoldingPosition = 3*));
				(*
				FOR i:=LOWER_BOUND(suctions, 1) TO UPPER_BOUND(suctions, 1) BY 1 DO
					
					IF i < UPPER_BOUND(suctions, 1)/2 THEN
						suctions[i].enable := robot.materialAtHoldingPosition = 2; //enable upper half suctions
					ELSE
						suctions[i].enable := robot.materialAtHoldingPosition = 3; //enable lower half suctions
					END_IF

				END_FOR
				*)
		END_CASE
		
		suctionTimer(IN:= , PT:= suctionDelay, Q=> , ET=> );
		suctionTimer.IN := TRUE;
		IF NOT suctionTimer.Q THEN
			RETURN;
		END_IF
		
		IF robot.Done THEN
			suctionTimer.IN := FALSE;
			loadStep := COMPLETE;
			RETURN;
		END_IF
		
		robot.setGroup(group := 9, value := robot.materialAtHoldingPosition);
	
	COMPLETE:
		robot.clearCommand();
		
		//check insertion quality
		suctionTimer(IN:= , PT:= suctionDelay, Q=> , ET=> );
		suctionTimer.IN := TRUE;
		IF NOT suctionTimer.Q THEN
			RETURN;
		END_IF
		
		IF InsertionQuality(suctions := suctions, insertionMaterial := loadedMaterials[surfaceID], recipeMaterial := material) THEN
			loadingSequence := TRUE;
		ELSE //recovery - restage a new bunk to <slot> and reload
			suctionTimer.IN := FALSE;
			loadStep := 100;
			
		END_IF
		
	100: //recovery - restage and reload
		CASE surfaceID OF
			Surface.TOP, Surface.LEFT:
				recoveryMagazine REF= magazineLeft;			
				recoveryStageStep REF= stageStepLeft;
				
			Surface.RIGHT, Surface.BOTTOM:
				recoveryMagazine REF= magazineRight;			
				recoveryStageStep REF= stageStepRight;
				
		END_CASE
		
		IF
			stageSingle(
				robot:= robot, 
				table:= table, 
				magazine:= recoveryMagazine, 
				stageStep:= recoveryStageStep, 
				slot:= slot, 
				material:= material, 
				fail=> fail)
		THEN
			SetSuctions(suctionPads := suctions, state := FALSE);
			loadStep := 0; //retry
		END_IF
	
END_CASE
END_METHOD

METHOD splitCombinedMaterials : BOOL
VAR_IN_OUT
	materialID : STRING;
	splitMaterial : STRING;
END_VAR
VAR
	i : INT;
END_VAR
FindAndSplitChar(
	sSeparatorChar:= '_', 
	pSrcString:= ADR(materialID), 
	
	pLeftString:= ADR(splitMaterial), 
	nLeftSize:= SIZEOF(splitMaterial), 
	
	pRightString:= ADR(materialID), 
	nRightSize:= SIZEOF(materialID), 
	
	bSearchFromRight:= FALSE);
END_METHOD

METHOD stage : BOOL
VAR_OUTPUT
	error : BOOL;
END_VAR
{warning disable C0371}

CASE stageSet OF
	0: //create staging template
		IF generateStagingTemplate() THEN
			stageSet := 10;
		END_IF
	
	10: //staging sequence
		IF
			stagingSequence(				
				robot:= robotLeft, 
				template:= stagingTemplateLeft,
				table:= stagingTableLeft,  
				magazine:= magazineLeft, 
				stageStep:= stageStepLeft, 
				iSlot:= iSlotLeft,
				error=> errorLeft)
			
			AND
			stagingSequence(
				robot:= robotRight, 
				template:= stagingTemplateRight, 
				table:= stagingTableRight, 
				magazine:= magazineRight, 
				stageStep:= stageStepRight, 
				iSlot:= iSlotRight,
				error=> errorRight)
		THEN
			stageStepLeft := stageStepRight := 0;
			iSlotLeft := iSlotRight := 0;
			
			stageSet := COMPLETE;
		END_IF
		
	COMPLETE:
		stagingTemplateRight.clear(); //clear the staging templates
		stagingTemplateLeft.clear();
		
		robotLeft.release(sectionID); //release the robots
		robotRight.release(sectionID);
		
		stageSet := 0;
		stage := TRUE;
		
END_CASE
END_METHOD

METHOD stageSingle : BOOL
VAR_IN_OUT
	robot : RobotA21;
	table : StagingTable;
	magazine : SkidMagazine;
	stageStep : INT;
END_VAR
VAR_INPUT
	slot : INT;
	material : STRING;
END_VAR
VAR_OUTPUT
	fail : BOOL;
END_VAR
VAR
	column : INT; //valid positions start from 1
END_VAR
VAR CONSTANT
	suctionDistance : INT := 10;
END_VAR
{warning disable C0371}
{warning disable C0195}
(*
this method allows the staging of single bunks without the use of a template
neccessary for restaging bunks that are not loaded properly into insertions
*)

IF
	material = '' OR_ELSE
	table.getSlot(i := slot) = material
THEN
	robot.clearCommand();
	stageSingle := TRUE;
	RETURN;
END_IF

//follow the template as is
CASE stageStep OF
	0:
		robot.clearCommand();
		IF robot.Ready THEN
			stageStep := 10;
		END_IF
		
	10: //grab from magazine
		IF NOT magazine.findSlot(materialID := material, atPosition => column) THEN
			fail := TRUE;
			RETURN;
		END_IF
		
		IF robot.eoatDistance < suctionDistance THEN //robot is grabbing material
			robot.HoldMaterial := magazine.getSlot(i := column);
		END_IF
		
		IF robot.Done THEN
			stageStep := COMPLETE;
			RETURN;
		ELSIF table.isOccupied(slot) THEN //wood bunk registered on table
			stageStep := 20;
			RETURN;
		END_IF
		
		robot.setGroup(group := 1, value := A21.STAGE_BUNK);
		robot.setGroup(group := 2, value := column);
		robot.setGroup(group := 3, value := slot);
	
	20: //place to table
		IF
			table.isOccupied(slot) AND //staging table slot is occupied
			table.getSlot(slot) = '' AND //staging table has not recorded a bunk
			robot.HoldMaterial <> '' //robot is carrying a bunk
		THEN //move material from robot to table
			table.place(i := slot, materialID := robot.HoldMaterial);
			robot.HoldMaterial := '';
		END_IF
		
		IF robot.Done THEN
			stageStep := COMPLETE;
			RETURN;
		END_IF
	
	COMPLETE: //check here if staging is successful or needs to be repeated
		//if the material is registered on the table, this step will not be evaluated due to the guard clause above
		robot.clearCommand();
		IF table.isOccupied(slot) AND table.getSlot(i := slot) = material THEN
			stageSingle := TRUE;
		ELSE
			stageStep := 0;
		END_IF
		
END_CASE
END_METHOD

METHOD stagingSequence : BOOL
VAR_IN_OUT
	robot : RobotA21;
	template : StagingTable;
	table : StagingTable;
	magazine : SkidMagazine;
	stageStep : INT;
	iSlot : INT;
END_VAR
VAR_OUTPUT
	error : BOOL;
END_VAR
VAR
	magazineColumn : INT; //valid positions start from 1
END_VAR
VAR CONSTANT
	(*
	WIP : INT := 0;
	PASSED : INT := 1;
	FAILED : INT := 2;
	*)
	suctionDistance : INT := 10;
END_VAR
VAR_STAT
	tempMaterial : STRING;
	tempOccupied : BOOL;
	temp : BOOL;
	
	adr1, adr2 : PVOID;
END_VAR
{warning disable C0371}
{warning disable C0195}
iSlot := MAX(1, iSlot); //ensures iSlot is at least 1

IF //staging table is full or matches staging template
	table.isFull() OR iSlot > 10 OR 
	MEMCMP(
		table.slots, 
		template.slots, 
		SIZEOF(table.slots^) * (1 + UPPER_BOUND(table.slots, 1) - LOWER_BOUND(table.slots, 1)) ) = 0
THEN
	robot.clearCommand();
	robot.release(sectionID);
	stagingSequence := TRUE;
	RETURN;
	
ELSIF template.getSlot(i := iSlot) = '' THEN
	iSlot := iSlot + 1;
	RETURN;
END_IF

IF robot.error THEN
	error := TRUE;
	RETURN;
ELSIF robot.reservation <> sectionID AND_THEN NOT robot.reserve(sectionID) THEN
	RETURN;
ELSIF robot.tool <> sectionID AND_THEN NOT robot.changeEOAT(targetTool := sectionID) THEN
	RETURN;
END_IF

//follow the template as is
IF
	stageSingle(
		robot:= robot, 
		table:= table, 
		magazine:= magazine, 
		stageStep:= stageStep, 
		slot:= iSlot, 
		material:= template.getSlot(iSlot), 
		fail=> error)
THEN
	iSlot := iSlot + 1;
	stageStep := 0;
END_IF
END_METHOD

ACTION stopSequence:
insertionLeft.stop();
insertionRight.stop();
pistonBottom.stop();

robotLeft.clearCommand();
robotRight.clearCommand();

//stop conveyors
END_ACTION

METHOD validateSuctionQuality : BOOL
VAR_INPUT
	checkTop : BOOL;
	checkLeft : BOOL;
	checkRight : BOOL;
	checkBottom : BOOL;
END_VAR
validateSuctionQuality := 
	(
		NOT checkTop OR_ELSE InsertionQuality(
			suctions:= suctionTop, 
			insertionMaterial:= loadedMaterials[Surface.TOP], 
			recipeMaterial:= materialsArr[iPair].top)
	) AND
	(
		NOT checkLeft OR_ELSE InsertionQuality(
			suctions:= suctionLeft, 
			insertionMaterial:= loadedMaterials[Surface.LEFT], 
			recipeMaterial:= materialsArr[iPair].left)
	) AND
	(
		NOT checkRight OR_ELSE InsertionQuality(
			suctions:= suctionRight, 
			insertionMaterial:= loadedMaterials[Surface.RIGHT], 
			recipeMaterial:= materialsArr[iPair].right)
	) AND
	(
		NOT checkBottom OR_ELSE InsertionQuality(
			suctions:= suctionBottom, 
			insertionMaterial:= loadedMaterials[Surface.BOTTOM], 
			recipeMaterial:= materialsArr[iPair].bottom)
	);
END_METHOD

END_FUNCTION_BLOCK
